(* IEC 61131-3 sources: Lasal/CPU_5344_V01/Class/Or_clientServer, 1 file *)

(* ---- Or_clientServer.st ---- *)
(*!
<Class
	Name               = "Or_clientServer"
	Revision           = "0.0"
	RealtimeTask       = "false"
	CyclicTask         = "false"
	BackgroundTask     = "false"
	Sigmatek           = "false"
	OSInterface        = "false"
	HighPriority       = "false"
	Automatic          = "false"
	UpdateMode         = "Prescan"
	SharedCommandTable = "true"
	Objectsize         = "(284,120)">
	<Channels>
		<Server Name="ClassSvr" Visualized="false" Initialize="false" WriteProtected="true" Retentive="false"/>
		<Server Name="Server" Visualized="false" Initialize="false" WriteProtected="false" Retentive="false"/>
		<Client Name="Client" Required="true" Internal="false"/>
	</Channels>
</Class>
*)
Or_clientServer : CLASS
  //Servers:
	ClassSvr 	: SvrChCmd_DINT;
	Server 	: SvrCh_DINT;
  //Clients:
	Client 	: CltCh_DINT;
  //Variables:
  //Functions:

	FUNCTION VIRTUAL GLOBAL ClassSvr::Read
		VAR_OUTPUT
			output (EAX) 	: DINT;
		END_VAR;
  //Tables:
	FUNCTION @STD
		VAR_OUTPUT
			ret_code	: CONFSTATES;
		END_VAR;
	FUNCTION GLOBAL TAB @CT_;
END_CLASS;

// Class Or_clientServer created by JdK at 21-5-2019 for standard lib MPS
// classsvr is made 1 if or client or server is 1, else it's 0

FUNCTION VIRTUAL GLOBAL Or_clientServer::ClassSvr::Read
	VAR_OUTPUT
		output (EAX) 	: DINT;
	END_VAR

  Client:=Client.Read();
  ClassSvr:=Client|Server;

	output := ClassSvr;

END_FUNCTION
